INTERFACE ITF_UtworzSzablonReceptury

METHOD Utworz : BOOL
VAR_INPUT
	stReceptury				: REFERENCE TO ST_Receptury;
END_VAR
END_METHOD

END_INTERFACE

(* stored: Version 1.1.0.1
   Itf ITF_UtworzSzablonReceptury: Id {b1567e56-d4df-0616-2298-2e3fa9712612}
   Method Utworz: Id {5c7b52e5-1d5a-0609-30f3-38875d3c12e4} *)
